TYPE ST_FeedbackWinch :
STRUCT
	l : REAL;
	l_t : REAL;
	l_tt : REAL;
END_STRUCT
END_TYPE

(* stored: Version 1.1.0.1, ProductVersion 3.1.4022.7
   DUT ST_FeedbackWinch: Id {2609b698-f679-4f88-a115-1cec61fc4353} *)
